FUNCTION getInUsint : USINT
VAR_INPUT
	bol_GlobalEnableForce		: BOOL;
	p_Input						: POINTER TO T_Ctrl_IoUsint;
END_VAR
VAR
END_VAR

(* Copyright 2017 Cimpress

Licensed under the Apache License, Version 2.0 (the "License");
you may not use this file except in compliance with the License.
You may obtain a copy of the License at

http://www.apache.org/licenses/LICENSE-2.0

Unless required by applicable law or agreed to in writing, software
distributed under the License is distributed on an "AS IS" BASIS,
WITHOUT WARRANTIES OR CONDITIONS OF ANY KIND, either express or implied.
See the License for the specific language governing permissions and
limitations under the License. *)

p_Input^.state := p_Input^.map;

IF (p_Input^.EnForce AND bol_GlobalEnableForce) THEN
	p_Input^.intern := p_Input^.force;
ELSE
	p_Input^.intern := p_Input^.map;
END_IF;

getInUsint := p_Input^.intern;

END_FUNCTION

(* stored: Version 1.1.0.1, ProductVersion 3.1.4019.2
   POU getInUsint: Id {d14befb2-e4e1-4e32-b4ed-195913a07eec}, SpecialFunc None *)
